// TIA Portal V16 export
// export: Created 2021-07-12T14:47:16.304552Z, ExportSetting WithDefaults, DisplayName Totally Integrated Automation Portal, DisplayVersion V16, DisplayName TIA Portal Version Control Interface, DisplayVersion V16, DisplayName TIA Portal Openness, DisplayVersion V16, DisplayName STEP 7 Professional, DisplayVersion V16, DisplayName STEP 7 Safety, DisplayVersion V16, DisplayName WinCC Professional, DisplayVersion V16
DATA_BLOCK "InstHydraulicsSimulationAnalog1"   // DB33160
{ DB_Accessible_From_OPC_UA := 'FALSE' }
FAMILY : SimaHydTO
VERSION : 1.0
// stored: AutoNumber true, DBAccessibleFromOPCUA false, InstanceOfName LSimaHydTO_HydraulicSimulationAnalog, InstanceOfType FB
"LSimaHydTO_HydraulicSimulationAnalog"
   // VAR_INPUT
   //    enable : Bool;
   //    analogInput : Int;
   //    initPosition : LReal;
   //    minPosition : LReal;
   //    maxPosition : LReal;
   //    maxVelocity : LReal;
   //    maxForce : LReal;
   //    springDistance : LReal;
   //    externalForce : LReal;
   //    dynamicFrictionFactor : LReal;
   //    fixedStop : LReal;
   //    fixedStopInverse : Bool;
   //    forceInverse : Bool;
   //    delayTime : LReal;
   //    cycleTime : UDInt;
   //    vChar_DB_NUMBER : UInt;
   //    axisTO : DB_ANY;
   //    Pozisyon_Input : LReal;
   // END_VAR
   // VAR_OUTPUT
   //    busy { ExternalWritable := 'False'} : Bool;
   //    active { ExternalWritable := 'False'} : Bool;
   //    error { ExternalWritable := 'False'} : Bool;
   //    status { ExternalWritable := 'False'} : Word;
   //    simulatedPosition { ExternalWritable := 'False'} : LReal;
   //    simulatedForce { ExternalWritable := 'False'} : LReal;
   //    simulatedVChar { ExternalWritable := 'False'} : UInt;
   //    forceSensorAnalog_A { ExternalWritable := 'False'} : Word;
   //    forceSensorAnalog_B { ExternalWritable := 'False'} : Word;
   // END_VAR
   // VAR_IN_OUT
   //    tel81in : PD_TEL81_IN;
   //    tel81out : PD_TEL81_OUT;
   // END_VAR
   // VAR
   //    statSetPoint { ExternalAccessible := 'False'; ExternalVisible := 'False'; ExternalWritable := 'False'} : LReal;
   //    statVelSetPoint { ExternalAccessible := 'False'; ExternalVisible := 'False'; ExternalWritable := 'False'} : LReal;
   //    statActualVChar { ExternalAccessible := 'False'; ExternalVisible := 'False'; ExternalWritable := 'False'} : UInt;
   //    statSampleTime { ExternalAccessible := 'False'; ExternalVisible := 'False'; ExternalWritable := 'False'} : LReal;
   //    statActualPosition { ExternalAccessible := 'False'; ExternalVisible := 'False'; ExternalWritable := 'False'} : LReal;
   //    statActualForce { ExternalAccessible := 'False'; ExternalVisible := 'False'; ExternalWritable := 'False'} : LReal;
   //    statForceFactor { ExternalAccessible := 'False'; ExternalVisible := 'False'; ExternalWritable := 'False'} : LReal;
   //    statEnableOld { ExternalAccessible := 'False'; ExternalVisible := 'False'; ExternalWritable := 'False'} : Bool;
   //    instSetPointPT1 { ExternalAccessible := 'False'; ExternalVisible := 'False'; ExternalWritable := 'False'; S7_SetPoint := 'True'} : "LSimaHydTO_T1";
   //    statPosLimitForce { ExternalAccessible := 'False'; ExternalVisible := 'False'; ExternalWritable := 'False'} : LReal;
   //    statNegLimitForce { ExternalAccessible := 'False'; ExternalVisible := 'False'; ExternalWritable := 'False'} : LReal;
   //    statFrictionForce { ExternalAccessible := 'False'; ExternalVisible := 'False'; ExternalWritable := 'False'} : LReal;
   //    instSimpleEncSetValue { ExternalAccessible := 'False'; ExternalVisible := 'False'; ExternalWritable := 'False'; S7_SetPoint := 'True'} : "LSimaHydTO_SimpleEncTel81";
   //    statVCharDB { ExternalAccessible := 'False'; ExternalVisible := 'False'; ExternalWritable := 'False'} : DB_ANY;
   //    statErrorVariant { ExternalAccessible := 'False'; ExternalVisible := 'False'; ExternalWritable := 'False'} : Int;
   //    statIntVelocityFactor { ExternalAccessible := 'False'; ExternalVisible := 'False'; ExternalWritable := 'False'} : LReal;
   // END_VAR
BEGIN
END_DATA_BLOCK
